FUNCTION_BLOCK FB_Btn
VAR_INPUT
	xStart:BOOL;
	xStop:BOOL;
	xReset:BOOL;
	xNextPas:BOOL;
	xAru:BOOL;
	
	xManAct1Rentre: BOOL;
	xManAct1Sort : BOOL;
	
	xManAct2Rentre: BOOL;
	xManAct2Sort : BOOL;
	
	xManAct3Rentre: BOOL;
	xManAct3Sort : BOOL;
END_VAR
VAR_OUTPUT
END_VAR
VAR
END_VAR

END_FUNCTION_BLOCK

(* stored: Version 1.1.0.1, ProductVersion 3.1.4020.6
   POU FB_Btn: Id {339910d3-7b2d-46d2-b617-7a7170002754}, SpecialFunc None *)
